FUNCTION WRITE_PROTECTED_DINT
VAR_INPUT
    Ptr : POINTER TO DINT;
    Value : DINT;
END_VAR

Ptr^ := Value;

END_FUNCTION

(* stored: Version 1.1.0.1, ProductVersion 3.1.4022.18
   POU WRITE_PROTECTED_DINT: Id {e753c22d-5f40-4162-b951-1bab50066302}, SpecialFunc None *)
